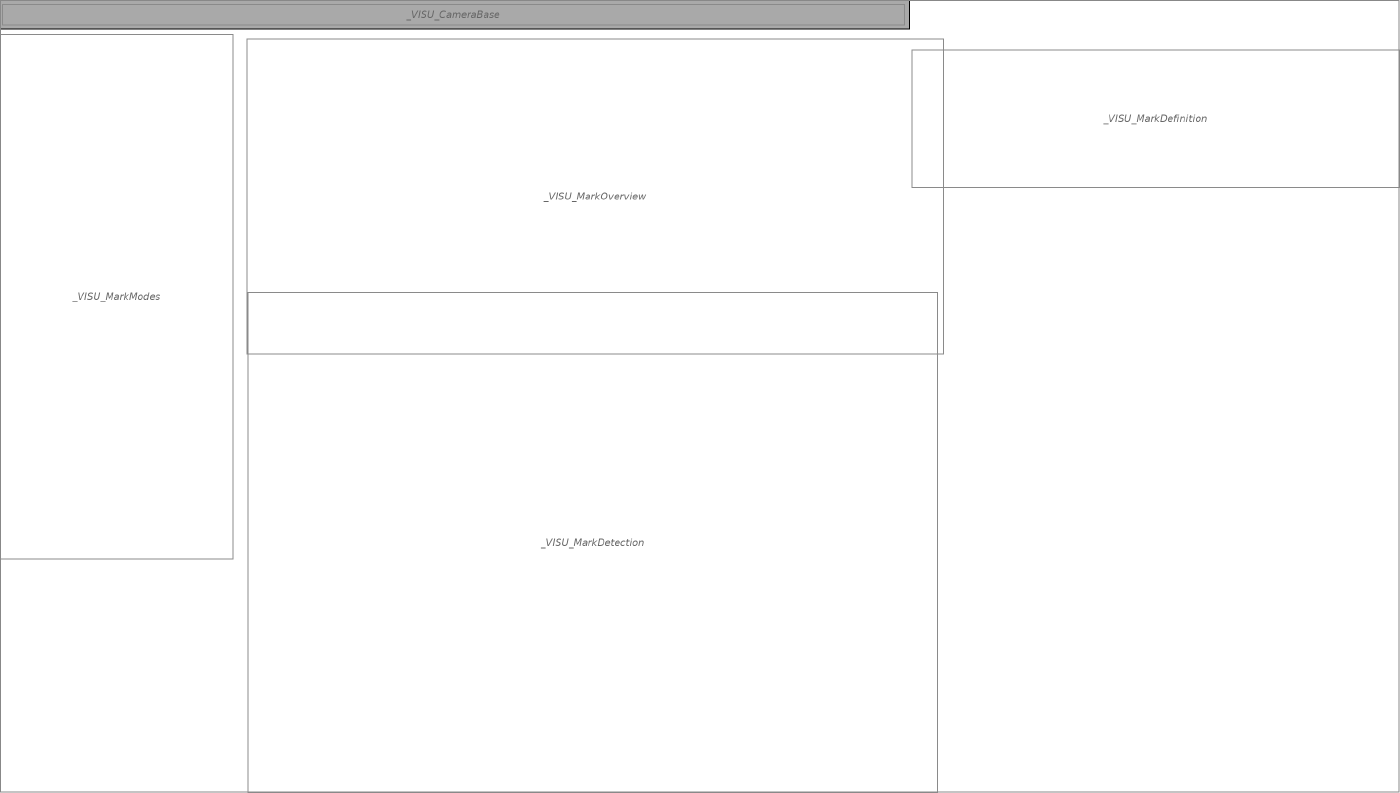
VISUALIZATION _VISU_MarkCamera_WEU  // 1447x820
VAR_IN_OUT
  mInst : FB_MarkCamera_WEU;
END_VAR
    RoundedRectangle (0,0 940x30)
    Frame (255,40 720x326)
        shows _VISU_MarkOverview(mInst := mInst)
    Frame (2,4 933x22)
        shows _VISU_CameraBase(m_Inst := mInst)
    Frame (0,35 241x543)
        shows _VISU_MarkModes(mInst := mInst)
    Frame (256,302 713x518)
        shows _VISU_MarkDetection(mInst := mInst.fbMarkDetection)
    Frame (942,51 505x143)
        shows _VISU_MarkDefinition(mInst := mInst.fbMarkDefinition)
END_VISUALIZATION

(* stored: Version 1.1.0.1, ProductVersion 3.1.4024.11
   Visu _VISU_MarkCamera_WEU: Id {daf9130b-ea3a-4d24-bb53-8b3f847e2ec5} *)
